INTERFACE I_NodePrototype EXTENDS I_Serializable

METHOD Clone : I_Node
VAR_INPUT
END_VAR
END_METHOD

END_INTERFACE

(* stored: Version 1.1.0.1, ProductVersion 3.1.4024.12
   Itf I_NodePrototype: Id {80358c56-c17b-4fd6-bd4f-d40c394564e4}
   Method Clone: Id {f434dfaa-76a7-4368-a9ea-37c90c5fda5f} *)
